TYPE (* DataPanel Modules with low IO density DO Struct + Source Address *)
  (* Version 1.1, 2026-05-28, franz *)
  PACKAGE DataPanel::io::LO::DQ;
  IMPORT eclipse4diac::core::TypeHash;
  IMPORT DataPanel::io::LO::const::LO::LO_00;
  IMPORT DataPanel::io::LO::DQ::DataPanel_LO_DO_S;
  IMPORT DataPanel::io::LO::DQ::DataPanel_LO_DO::InvalidL;
  DataPanel_LO_DO_S_Octal_SA : STRUCT
    u8SAMember : USINT := LO_00; (* Node SA 217..224 *)
    Port1 : DataPanel::io::LO::DQ::DataPanel_LO_DO_S := InvalidL; (* Identify the Port 1A..4B *)
    Port2 : DataPanel::io::LO::DQ::DataPanel_LO_DO_S := InvalidL; (* Identify the Port 1A..4B *)
    Port3 : DataPanel::io::LO::DQ::DataPanel_LO_DO_S := InvalidL; (* Identify the Port 1A..4B *)
    Port4 : DataPanel::io::LO::DQ::DataPanel_LO_DO_S := InvalidL; (* Identify the Port 1A..4B *)
    Port5 : DataPanel::io::LO::DQ::DataPanel_LO_DO_S := InvalidL; (* Identify the Port 1A..4B *)
    Port6 : DataPanel::io::LO::DQ::DataPanel_LO_DO_S := InvalidL; (* Identify the Port 1A..4B *)
    Port7 : DataPanel::io::LO::DQ::DataPanel_LO_DO_S := InvalidL; (* Identify the Port 1A..4B *)
    Port8 : DataPanel::io::LO::DQ::DataPanel_LO_DO_S := InvalidL; (* Identify the Port 1A..4B *)
  END_STRUCT;
END_TYPE
